# EPICS autosave request: soft_iocs/meas_comp/meas_compApp/Db/calc_settings.req
# FILE... calc_settings.req
# USAGE.. calc Record fields autosave'd.
$(P).A
$(P).B
$(P).C
$(P).D
$(P).E
$(P).F
$(P).G
$(P).H
$(P).I
$(P).J
$(P).K
$(P).L
$(P).INPA
$(P).INPB
$(P).INPC
$(P).INPD
$(P).INPE
$(P).INPF
$(P).INPG
$(P).INPH
$(P).INPI
$(P).INPJ
$(P).INPK
$(P).INPL
$(P).CALC$
$(P).SCAN
$(P).PREC
$(P).FLNK
$(P).DESC
$(P).EGU
